{attribute 'reflection'} 
FUNCTION_BLOCK FB_WorkerDefGrid_Python EXTENDS FB_WorkerDefGrid
VAR_INPUT
END_VAR
VAR_OUTPUT
END_VAR
VAR
  // interface to py script
  fbPythonInterface : FB_PythonInterface;
  
  // local copy of setttings
  _bNewJob : BOOL;  // new job was activated
  _CamGridSettings : ST_CameraGridSettings;
  _DefGridSettings : ST_DefGridSettings;
END_VAR

VAR CONSTANT
  fC_DEFAULT_WOKER_POSITION : LREAL := 0.01;      // default worker position in [m]
END_VAR

METHOD PROTECTED  Attach : BOOL
VAR_INPUT
  iCT              : I_CT;                         (*container at triggered event position*)
END_VAR
VAR
  sCamSettings : ST_CameraGridSettings;
END_VAR
Attach := FALSE;
IF SUPER^.Attach(iCT:=iCT) THEN
  // OK, attached (enabled, was ok to be attached)
  
  // setup check
  IF _pParamMediator = 0 THEN Release(iCT:=iCT); LogError('Invalid param mediator'); RETURN; END_IF
  
  // Additional worker checks
  // - do we have a valid job? used mode?
  IF _CamGridSettings.eCameraMode > E_CameraMode.NoCorrection AND (_pAttachedCt^.pJob = 0 OR NOT _bJobActive) THEN
    _pAttachedCt^.AbortDeformation(sReason:='No valid job', Src:=_pEcSrc^);
     Release(iCT:=iCT);
     
  ELSIF _CamGridSettings.eCameraMode > E_CameraMode.NoCorrection THEN
    // OK attach
    // -- only create ct if a deformation is active
    IF CreateDefCt(iCT:=iCT) THEN
        // set state
        _pAttachedCt^.StartDeformation(eDeformationStep:=E_DeformationStep.createdScriptContainer);
        // attached
        Attach := TRUE;
    END_IF
  ELSE
    ; // ignore attach
  END_IF
ELSE
  // parent attach failed
END_IF
END_METHOD

(*
  Create/Release virtual ct in deformation handlers.
  :return: TRUE if success
*)
METHOD PRIVATE CreateDefCt : BOOL;
VAR_INPUT
  iCT : I_CT;
END_VAR
IF iCT = 0 THEN RETURN; END_IF

IF _CamGridSettings.eCameraMode >= E_CameraMode.Live THEN
  IF fbPythonInterface.RegisterCT(iCT.pCT^.nMemIndex) THEN
    CreateDefCt := TRUE;
  ELSE
    _pAttachedCt^.AbortDeformation(sReason:='Could not register to script', Src:=_pEcSrc^);
  END_IF
ELSE
  CreateDefCt := TRUE;
END_IF
END_METHOD

(*
  Delete/Release virtual ct in deformation handlers.
  :return: TRUE if sucess
*)
METHOD DeleteDefCt : BOOL
VAR_INPUT
  iCT : I_CT;
END_VAR
IF iCT = 0 THEN RETURN; END_IF

IF _CamGridSettings.eCameraMode >= E_CameraMode.Live THEN
  IF fbPythonInterface.RemoveCT(iCT.pCT^.nMemIndex) THEN
    DeleteDefCt := TRUE;
  ELSE
    LogError('Could not delete ct in script');
  END_IF
END_IF
END_METHOD

METHOD InitWorkerPython
VAR_INPUT
  aScriptPath : T_MaxString;                     // path to cmd scripts
  //aAmsLocalHost : T_AmsNetID;                    // Ams netId localhost of the pc to run the script 
END_VAR
IF NOT bInitialized OR _pCtManager = 0 THEN LogError('Base Worker not initialized! call init() before'); RETURN; END_IF

// worker specific init

fbPythonInterface.Init(
  sCTManagerPath := _pCtManager^.sCTDefGridInstancesPath, 
  sScriptPath:=aScriptPath
);
END_METHOD

METHOD mJobStart
VAR_INPUT
	sJobDef	: CalmarCompPrint.I_JobDefinition;
END_VAR
// checks and fix defaults
IF _pParamMediator = 0 THEN LogError('JobStart: invalid parameter configuration'); RETURN; END_IF
IF _fWorkerPosition = 0 THEN _fWorkerPosition := fC_DEFAULT_WOKER_POSITION; LogError(F_Concat3(_name, ': worker position not set, set default=', TO_STRING(fC_DEFAULT_WOKER_POSITION))); END_IF

// configure
_fImageDepthM := sJobDef.fImageDepth/1000;
_fImageWidthM := sJobDef.fImageWidth/1000;
_fCtSecurityReleasePos := F_MeterToSubPixel(fPosMeter:=_fImageDepthM + fC_MIN_SHEET_GAP, fResoSubPx:=_fPrintResolution*_fSubPxResolution);

_bNewJob := TRUE;
_bJobActive := TRUE;
END_METHOD

METHOD  mJobStop
VAR_INPUT
	sStatus	: CalmarCompPrint.I_JobStatus;
END_VAR
fbPythonInterface.JobStop();
_bJobActive := FALSE;
END_METHOD

METHOD  work
VAR_INPUT
END_VAR
VAR
  i : UDINT;
  tempCt  : POINTER TO FB_ContainerDefGrid;
  bDeformationDone : BOOL;
  bDeformationError : BOOL;
  nConvErr : UDINT;
  rT_EnablePyIf  : R_TRIG;
END_VAR
SUPER^.work();

IF _pParamMediator <> 0 THEN
   // -- get latest camera & deformation settings
  _CamGridSettings := _pParamMediator^.sCameraGridSettings;
  _DefGridSettings := _pParamMediator^.sDeformationGridSetttings;
END_IF

IF _bNewJob OR rT_EnablePyIf.Q THEN   // new job activated or ente
  _bNewJob := FALSE;
  
  // setup script
  fbPythonInterface.JobStart(
    nJobImageWidth:=DINT_TO_UDINT(F_MeterToSubPixel(fPosMeter:=_fImageDepthM, fResoSubPx:=_fPrintResolution)),
    nJobImageHeigth:=DINT_TO_UDINT(F_MeterToSubPixel(fPosMeter:=_fImageWidthM, fResoSubPx:=_fPrintResolution)),
    nCamFrameWidth:=DINT_TO_UDINT(FC_LREAL_TO_DINT(_CamGridSettings.fGridFeaturePitch, ADR(nConvErr))),
    pGridSettings:=ADR(_DefGridSettings)
  );
END_IF

// start/stop script
IF _CamGridSettings.eCameraMode >= E_CameraMode.Live AND THIS^.bEnable THEN 
  fbPythonInterface.bEnable := TRUE;
ELSE
  fbPythonInterface.bEnable := FALSE;
END_IF
rT_EnablePyIf(CLK:=fbPythonInterface.bEnable);

fbPythonInterface();

IF _pAttachedCt <> 0 THEN
  // nothing to do anymore just release CT
  // NOTE: the delete of the CT is done by DeleteDefCt() method directly into fbPythonInterface
  Release(_pAttachedCt^);
END_IF
END_METHOD

END_FUNCTION_BLOCK

(* stored: Version 1.1.0.1, ProductVersion 3.1.4024.3
   POU FB_WorkerDefGrid_Python: Id {da715aa5-d637-40ab-8d33-e404e3b6a6f1}, SpecialFunc None
   Method Attach: Id {42eaf325-ff4e-48df-be91-9b20bce3da44}
   Method CreateDefCt: Id {bdf419b5-1889-4837-99cf-ef4a36422f29}
   Method DeleteDefCt: Id {1250acd3-857f-4045-a296-4dd4aaa257e9}
   Method InitWorkerPython: Id {343b3a60-1392-4b26-a0f9-056258434c15}
   Method mJobStart: Id {0fd0f7ed-3d4d-47aa-ba8e-6404bd51c209}
   Method mJobStop: Id {db89a0b9-8d28-4bf7-9778-94d597d27cae}
   Method work: Id {3c4c9ab8-eeba-4bde-9db0-7737c05146ce} *)
